FUNCTION F_MultiplicationFunction : REAL
VAR_INPUT
	rInput1 : REAL;
	rInput2 : REAL;
END_VAR
VAR
END_VAR

F_MultiplicationFunction := rInput1 * rInput2;

END_FUNCTION

(* stored: Version 1.1.0.1, ProductVersion 3.1.4024.13
   POU F_MultiplicationFunction: Id {b85837a6-db27-4059-9821-fe8e5465b2fb}, SpecialFunc None *)
